FUNCTION_BLOCK centralServer (* Basic Function Block Type *)
  (* Standard: 61499-2 *)
  (* Version 0.2, 2003-12-04, JHC, Rockwell Automation, Renamed for better indexing. *)
  (* Version 0.1, 2002-11-05, JHC, Rockwell Automation, Corrected missing ST element in Algorithm REQ. *)
  (* Version 0.0, 2000-05-30, JHC, Rockwell Automation *)
  (* Compiler header: package fb.rt.cs725; *)
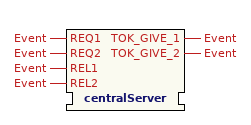
  EVENT_INPUT
    REQ1;
    REQ2;
    REL1;
    REL2;
  END_EVENT
  EVENT_OUTPUT
    TOK_GIVE_1;
    TOK_GIVE_2;
  END_EVENT
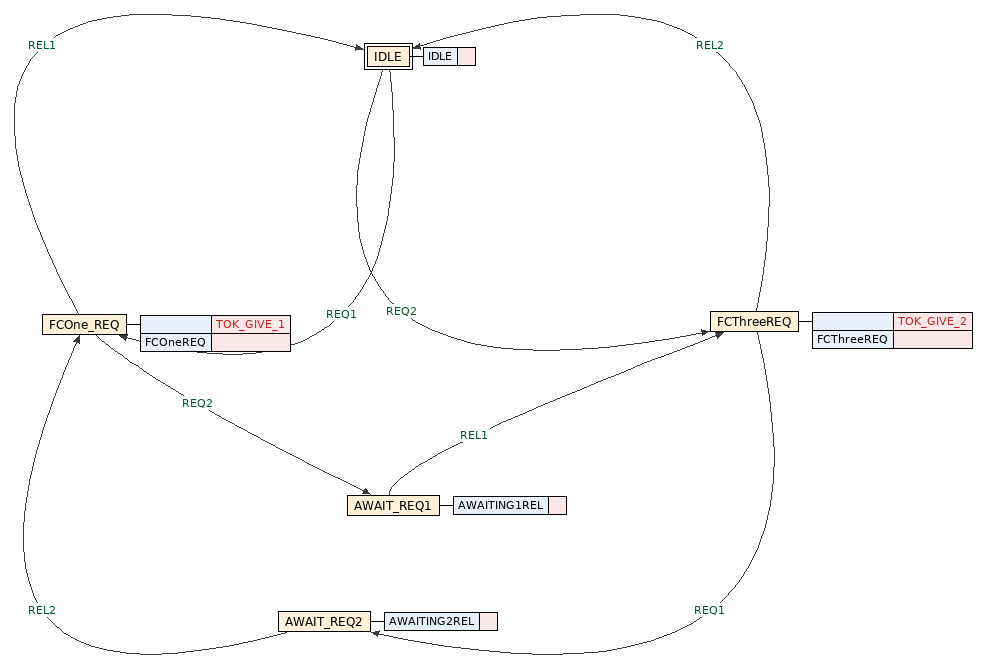
  EC_STATES
    IDLE : IDLE; (* Initial State *)
    FCOne_REQ : -> TOK_GIVE_1, FCOneREQ;
    FCThreeREQ : -> TOK_GIVE_2, FCThreeREQ;
    AWAIT_REQ1 : AWAITING1REL;
    AWAIT_REQ2 : AWAITING2REL;
  END_STATES
  EC_TRANSITIONS
    IDLE TO FCThreeREQ := REQ2;
    IDLE TO FCOne_REQ := REQ1;
    FCThreeREQ TO IDLE := REL2;
    FCOne_REQ TO IDLE := REL1;
    FCOne_REQ TO AWAIT_REQ1 := REQ2;
    AWAIT_REQ1 TO FCThreeREQ := REL1;
    FCThreeREQ TO AWAIT_REQ2 := REQ1;
    AWAIT_REQ2 TO FCOne_REQ := REL2;
  END_TRANSITIONS
  ALGORITHM IDLE IN Java:

  END_ALGORITHM
  ALGORITHM FCThreeREQ IN Java:

  END_ALGORITHM
  ALGORITHM FCOneREQ IN Java:

  END_ALGORITHM
  ALGORITHM AWAITING1REL IN Java:

  END_ALGORITHM
  ALGORITHM AWAITING2REL IN Java:

  END_ALGORITHM
END_FUNCTION_BLOCK
